Staubli VAL3: EnterPageKey.pgx

program EnterPageKey(num& x_nKey, num& x_nSelect, string& x_sItem)
  local string l_sStr
  local num l_nKey
  local string l_sEmpty
  local string l_sValue
  local num l_nItem
  local num l_nView
  local string l_sItem
  local point lp
  local string l_sYN[2]
  local bool l_bRes
  local num l_nTemp
begin
  //
  //编辑项目
  switch x_nSelect
    //X
    case 0
      if x_nKey==270
        call user:editNum(x_sItem,sListItemValue[x_nSelect],prd:pDemo[nSelected].trsf.x,x_nSelect)
      endIf
    break
    //Y
    case 1
      if x_nKey==270
        call user:editNum(x_sItem,sListItemValue[x_nSelect],prd:pDemo[nSelected].trsf.y,x_nSelect)
      endIf
    break
    //Z
    case 2
      if x_nKey==270
        call user:editNum(x_sItem,sListItemValue[x_nSelect],prd:pDemo[nSelected].trsf.z,x_nSelect)
      endIf
    break
    //rx
    case 3
      if x_nKey==270
        call user:editNum(x_sItem,sListItemValue[x_nSelect],prd:pDemo[nSelected].trsf.rx,x_nSelect)
      endIf
    break
    //ry
    case 4
      if x_nKey==270
        call user:editNum(x_sItem,sListItemValue[x_nSelect],prd:pDemo[nSelected].trsf.ry,x_nSelect)
      endIf
    break
    //rz
    case 5
      if x_nKey==270
        call user:editNum(x_sItem,sListItemValue[x_nSelect],prd:pDemo[nSelected].trsf.rz,x_nSelect)
      endIf
    break
    //PIn1
    case 6
      if x_nKey==270
        call SparePoint:setPoint(sListItemValue[x_nSelect])
        call SparePoint:start()
        call SparePoint:getPoint(sListItemValue[x_nSelect])
        x_sItem="PIn1     :"+sListItemValue[x_nSelect]
      endIf

    break
    //PIn2
    case 7
      if x_nKey==270
        call SparePoint:setPoint(sListItemValue[x_nSelect])
        call SparePoint:start()
        call SparePoint:getPoint(sListItemValue[x_nSelect])
        x_sItem="PIn2     :"+sListItemValue[x_nSelect]
      endIf
    break
    //POut1
    case 8
      if x_nKey==270
        call SparePoint:setPoint(sListItemValue[x_nSelect])
        call SparePoint:start()
        call SparePoint:getPoint(sListItemValue[x_nSelect])
        x_sItem="POut     :"+sListItemValue[x_nSelect]
      endIf
    break
    //IO1
    case 9
      if x_nKey==270
        call IO:setIO(sListItemValue[x_nSelect])
        call IO:Main(1)
        call IO:getIO(sListItemValue[x_nSelect])
        //
        x_sItem="IO1      :"+sListItemValue[x_nSelect]
      endIf

    break
    //IO2
    case 10
      if x_nKey==270
        call IO:setIO(sListItemValue[x_nSelect])
        call IO:Main(1)
        call IO:getIO(sListItemValue[x_nSelect])
        //
        x_sItem="IO2      :"+sListItemValue[x_nSelect]
      endIf
    break
    //delay
    case 11
      if x_nKey==270
        call user:editNum(x_sItem,sListItemValue[x_nSelect],l_nTemp,x_nSelect)
      endIf
    break
  endSwitch
  if x_nKey==270
    bUserRefresh=true
    bListRefresh=true
  endIf
end
